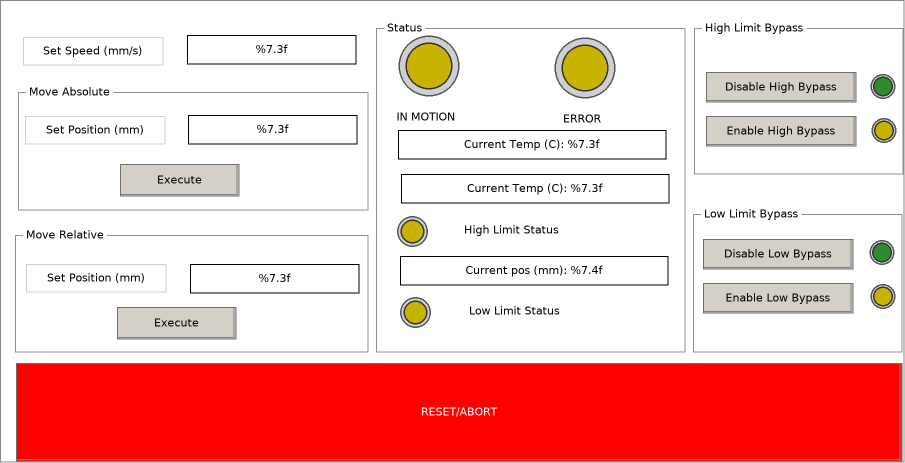
VISUALIZATION Visualization  // 905x463
    Rectangle (187,35 169x29), "%7.3f", text variable: MAIN.fSpeed
    Textfield (23,37 140x28), "Set Speed (mm/s)"
        OnMouseUp: write MAIN.fSpeed via Default, format %7.3f
    GroupBox (18,84 350x126), "Move Absolute"
        Button (102,80 119x32), "Execute"
            OnMouseUp: execute { MAIN.state:=E_State.moveAbs; }
        Rectangle (170,31 169x29), "%7.3f", text variable: MAIN.fPosition
        Textfield (7,32 140x28), "Set Position (mm)"
            OnMouseUp: write MAIN.fPosition via Default, format %7.3f
    GroupBox (15,227 353x125), "Move Relative"
        Button (102,80 119x32), "Execute"
            OnMouseUp: execute { MAIN.state:=E_State.moveRel; }
        Rectangle (175,37 169x29), "%7.3f", text variable: MAIN.fPosRel
        Textfield (11,37 140x28), "Set Position (mm)"
            OnMouseUp: write MAIN.fPosRel via Default, format %7.3f
    GroupBox (376,20 309x332), "Status"
        Lamp1 (18,11 70x70), variable: MAIN.M[1].axisRef.Status.Moving, style: Lamp-Lamp1-Yellow
        Label (6,82 88x30), "IN MOTION"
        Lamp1 (174,13 70x70), variable: MAIN.M[1].mcMoveAbs.Error or MAIN.M[1].mcMoveRel.Error or MAIN.M[1].mcReset.Error, style: Lamp-Lamp1-Yellow
        Label (162,84 88x30), "ERROR"
        Lamp1 (19,192 35x39), variable: not(MAIN.M[1].bLimHigh), style: Lamp-Lamp1-Yellow
        Label (67,195 137x30), "High Limit Status"
        Lamp1 (22,273 35x39), variable: not(MAIN.M[1].bLimLow), style: Lamp-Lamp1-Yellow
        Label (70,276 137x30), "Low Limit Status"
        Rectangle (24,236 268x29), "Current pos (mm): %7.4f", text variable: MAIN.M[1].axisRef.NcToPlc.ActPos
        Rectangle (22,110 268x29), "Current Temp (C): %7.3f", text variable: MAIN.Temp1
        Rectangle (25,154 268x29), "Current Temp (C): %7.3f", text variable: MAIN.Temp2
    Button (16,363 886x98), "RESET/ABORT"
        OnMouseUp: execute { Main.state:=E_State.reset; }
    Button (706,72 150x30), "Disable High Bypass"
        OnMouseDown: execute { MAIN.bHighBypass:=FALSE; }
    Button (706,116 150x30), "Enable High Bypass"
        OnMouseDown: execute { MAIN.bHighBypass:=TRUE; }
    Button (703,239 150x30), "Disable Low Bypass"
        OnMouseDown: execute { MAIN.bLowBypass:=FALSE; }
    Button (703,283 150x30), "Enable Low Bypass"
        OnMouseDown: execute { MAIN.bLowBypass:=TRUE; }
    Lamp1 (866,72 34x29), tooltip "Lim Enabled", variable: NOT MAIN.bHighBypass, style: Lamp-Lamp1-Green
    Lamp1 (867,116 34x29), tooltip "Lim Enabled", variable: MAIN.bHighBypass, style: Lamp-Lamp1-Yellow
    Lamp1 (865,238 34x29), tooltip "Lim Enabled", variable: NOT MAIN.bLowBypass, style: Lamp-Lamp1-Green
    Lamp1 (866,282 34x29), tooltip "Lim Enabled", variable: MAIN.bLowBypass, style: Lamp-Lamp1-Yellow
    GroupBox (694,20 209x154), "High Limit Bypass"
    GroupBox (693,206 209x146), "Low Limit Bypass"
END_VISUALIZATION

(* stored: Version 1.1.0.1, ProductVersion 3.1.4022.18
   Visu Visualization: Id {132d6d6e-87f6-4091-a481-5a0b7319f7f3} *)
